(* CODESYS project %VISU%Visualization_test.xml

Project tree, tasks and I/O mapping:
  visualisation Visualization_test
*)

// /Visualization_test
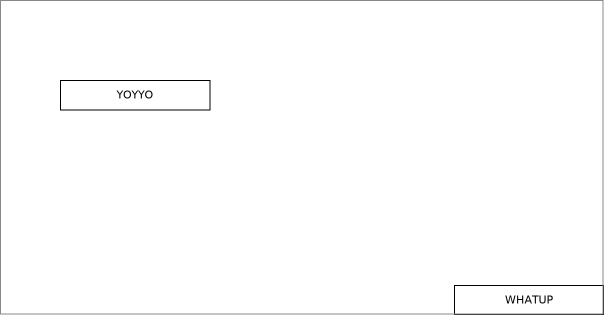
VISUALIZATION Visualization_test  // 604x315
    Rectangle (60,80 150x30), "YOYYO"
    Rectangle (454,285 150x30), "WHATUP"
END_VISUALIZATION
